(* CODESYS project Ergasia.project

Project tree, tasks and I/O mapping:
  Device : CODESYS Control Win V3, 3S - Smart Software Solutions GmbH, version 3.5.3.50
    application Application
      libraries: Standard, 3.5.2.0 (System)
      task MainTask (cyclic, interval t#20ms, priority 1) calls Main, Simulate
      task VISU_TASK (cyclic, interval 100 ms, priority 30) calls VisuElems.Visu_Prg
      program Main [SFC]: machine_check, Turn_off
      global variables GVL
      function block Flow_Control [SFC]: try_load, reset
      program Simulate [ST]
      visualisation Visualization
  text list GlobalTextList
  GlobalImagePool
*)

// Device/Application/GVL
VAR_GLOBAL
	start_switch: BOOL;
	stop_switch: BOOL;
	load_bottle: BOOL;
	water_filler: BOOL;
	water_filler_time: LREAL := 5;
	water_filler_end: BOOL;
	wf_elapsed: LREAL;
	bottle_position: LREAL;
	water_filler_lens: BOOL;
	capper_lens: BOOL;
	tagger_lens: BOOL;
	storing_bank_lens: BOOL := FALSE;
	corridor_moving: BOOL;
	capper_end: BOOL;
	tagger_time: LREAL := 3;
	tagger_end: BOOL;
	capper: BOOL;
	tagger: BOOL;
	capper_elapsed: LREAL;
	tagger_elapsed: LREAL;
	capper_time: LREAL := 2;
	stop_button: BOOL := FALSE;
	bottle_number: INT := 0;
	supplying_bank_lens: BOOL := TRUE;
	stbl_on_time: LREAL := 0;
	alarm: BOOL := FALSE;
	running: BOOL;
	full_supplying_bank: BOOL := FALSE;
	finished_bottles: INT := 0;
END_VAR

// Device/Application/Main
PROGRAM Main
VAR
	succ_check: BOOL;
END_VAR

VAR
	Flow_Control: Flow_Control;
END_VAR

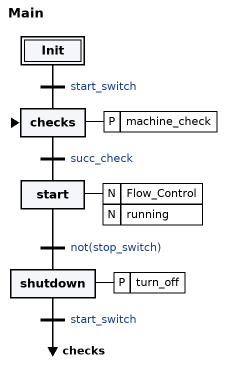
INITIAL_STEP Init:
END_STEP
TRANSITION FROM Init TO checks
    := start_switch;
END_TRANSITION
STEP checks:
    machine_check(P);
END_STEP
TRANSITION FROM checks TO start
    := succ_check;
END_TRANSITION
STEP start:
    Flow_Control(N);
    running(N);
END_STEP
TRANSITION FROM start TO shutdown
    := not(stop_switch);
END_TRANSITION
STEP shutdown:
    turn_off(P);
END_STEP
TRANSITION FROM shutdown TO checks
    := start_switch;
END_TRANSITION

ACTION machine_check:
IF (NOT(corridor_moving) AND NOT(water_filler) AND NOT(capper) AND NOT(tagger)) THEN
	succ_check := TRUE;
END_IF
END_ACTION

ACTION Turn_off:
(* calculate remaining time of operations *)
(*water_filler_time := water_filler_time - wf_elapsed;
capper_time := capper_time - capper_elapsed;
tagger_time := tagger_time - tagger_elapsed;*)
(*shut down machines *)
corridor_moving := FALSE;
water_filler := FALSE;
capper := FALSE;
tagger := FALSE;
succ_check := FALSE;
END_ACTION

END_PROGRAM

// Device/Application/Flow_Control
FUNCTION_BLOCK Flow_Control
VAR_INPUT
END_VAR
VAR_OUTPUT
END_VAR
VAR
END_VAR

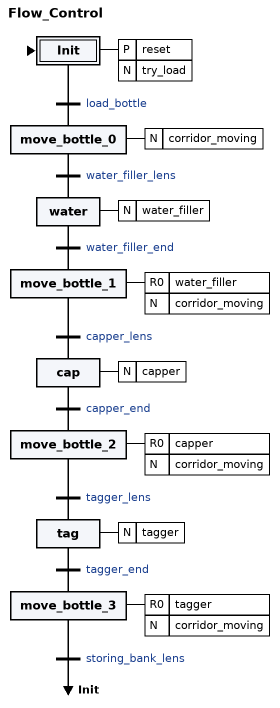
INITIAL_STEP Init:
    reset(P);
    try_load(N);
END_STEP
TRANSITION FROM Init TO move_bottle_0
    := load_bottle;
END_TRANSITION
STEP move_bottle_0:
    corridor_moving(N);
END_STEP
TRANSITION FROM move_bottle_0 TO water
    := water_filler_lens;
END_TRANSITION
STEP water:
    water_filler(N);
END_STEP
TRANSITION FROM water TO move_bottle_1
    := water_filler_end;
END_TRANSITION
STEP move_bottle_1:
    water_filler(R0);
    corridor_moving(N);
END_STEP
TRANSITION FROM move_bottle_1 TO cap
    := capper_lens;
END_TRANSITION
STEP cap:
    capper(N);
END_STEP
TRANSITION FROM cap TO move_bottle_2
    := capper_end;
END_TRANSITION
STEP move_bottle_2:
    capper(R0);
    corridor_moving(N);
END_STEP
TRANSITION FROM move_bottle_2 TO tag
    := tagger_lens;
END_TRANSITION
STEP tag:
    tagger(N);
END_STEP
TRANSITION FROM tag TO move_bottle_3
    := tagger_end;
END_TRANSITION
STEP move_bottle_3:
    tagger(R0);
    corridor_moving(N);
END_STEP
TRANSITION FROM move_bottle_3 TO Init
    := storing_bank_lens;
END_TRANSITION

ACTION try_load:
IF bottle_number > 0 AND supplying_bank_lens = TRUE THEN
	load_bottle := TRUE;
ELSE
	load_bottle := FALSE;
END_IF
END_ACTION

ACTION reset:
water_filler_end := FALSE;
capper_end := FALSE;
tagger_end := FALSE;
bottle_position := 0;
END_ACTION

END_FUNCTION_BLOCK

// Device/Application/Simulate
PROGRAM Simulate
VAR
END_VAR

(* initially closed switch simulation *)
stop_switch := NOT(stop_button);

(* completed bottle_number bottles simulation *)
IF bottle_number = 0 AND running THEN
	stop_button := TRUE;
END_IF

(* empty supplying bank simulation *)
IF supplying_bank_lens = FALSE AND bottle_position = 0 AND bottle_number > 0 THEN
	stop_button := TRUE;
	alarm := TRUE;
END_IF
IF supplying_bank_lens = TRUE AND bottle_position = 0 AND bottle_number > 0 THEN
	stop_button := FALSE;
	alarm := FALSE;
END_IF

(* full storing bank simulation *)
IF storing_bank_lens = TRUE AND full_supplying_bank THEN
	storing_bank_lens := TRUE;
ELSIF storing_bank_lens = TRUE AND NOT(full_supplying_bank) THEN
	storing_bank_lens := FALSE;
	stop_button := FALSE;
	alarm := FALSE;
	stbl_on_time := 0;
END_IF
IF storing_bank_lens = TRUE AND bottle_number > 0 THEN
	stbl_on_time := stbl_on_time + 0.02;
	IF stbl_on_time >= 2 THEN (* 2s lens on - arbitrary value *)
		stop_button := TRUE;
		alarm := TRUE;
	END_IF
END_IF

(* bottle moving in corridor simulation *)
IF (corridor_moving) THEN
	wf_elapsed := 0;
	capper_elapsed := 0;
	tagger_elapsed := 0;
	water_filler_lens := FALSE;
	capper_lens := FALSE;
	tagger_lens := FALSE;
	bottle_position := bottle_position + 0.015;
	IF bottle_position >=3 AND bottle_position <3.1 THEN
		water_filler_lens := TRUE;
		bottle_position := 3.2;
	ELSIF bottle_position >=6.1 AND bottle_position <6.2 THEN
		capper_lens := TRUE;
		bottle_position := 6.2;
	ELSIF bottle_position >=9.2 AND bottle_position <9.3 THEN
		tagger_lens := TRUE;
		bottle_position :=9.3;
	ELSIF bottle_position >=12.3 AND bottle_position <12.4 THEN
		storing_bank_lens := TRUE;
		bottle_position := 12.4;
		bottle_number := bottle_number - 1; (* bottle is finished *)
		finished_bottles := finished_bottles + 1;
	END_IF
END_IF

(* watering machine simulation *)
IF (water_filler) THEN
	water_filler_lens := TRUE;
	wf_elapsed := wf_elapsed + 0.02; (* 20ms cycle *)
	IF wf_elapsed >= water_filler_time THEN
		water_filler_end := TRUE;
	END_IF
END_IF

(* capping machine simulation *)
IF (capper) THEN
	capper_lens := TRUE;
	capper_elapsed := capper_elapsed + 0.02; (* 20ms cycle *)
	IF capper_elapsed >= capper_time THEN
		capper_end := TRUE;
	END_IF
END_IF

(* tagging machine simulation *)
IF (tagger) THEN
	tagger_lens := TRUE;
	tagger_elapsed := tagger_elapsed + 0.02; (* 20ms cycle *)
	IF tagger_elapsed >= tagger_time THEN
		tagger_end := TRUE;
	END_IF
END_IF

END_PROGRAM

// Device/Application/Visualization
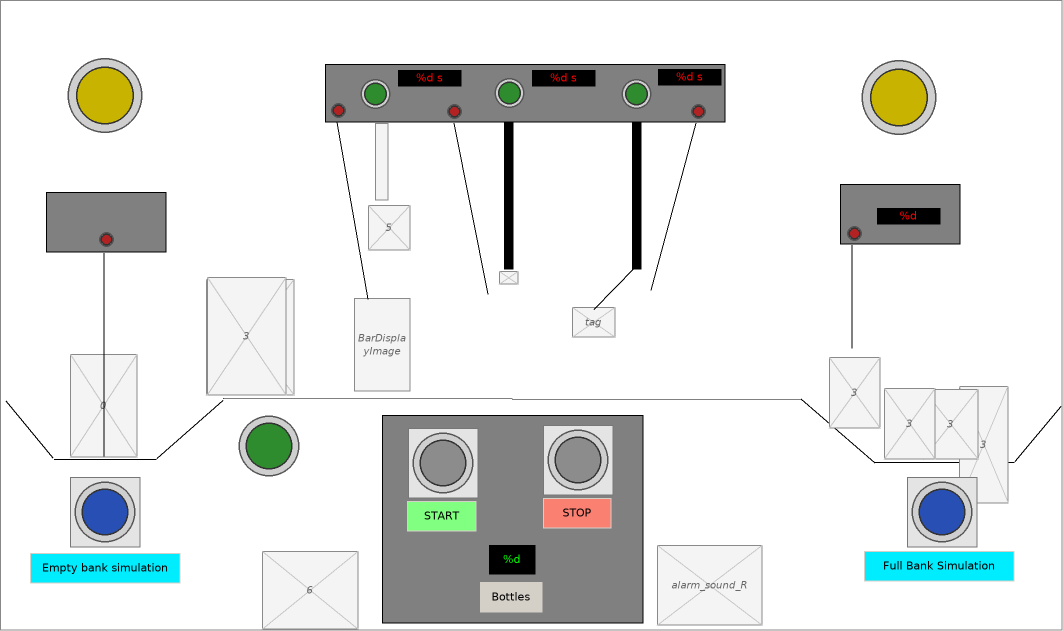
VISUALIZATION Visualization  // 1063x631
    Rectangle (382,415 261x208)
    PushSwitch (408,428 70x70), variable: start_switch, behaviour: TAP, style: Switch-PushSwitch-Gray
    PushSwitch (543,425 70x70), variable: stop_button, behaviour: TAP, style: Switch-PushSwitch-Gray
    Rectangle (489,545 46x29), "%d", text variable: bottle_number
        OnMouseDown: write the text variable via Edit, min 0, max 999
    Line (223,398) (801,399)
    Rectangle (325,64 400x58)
    BarDisplayImage (354,298 56x93), value: wf_elapsed, style: BarDisplayImage-Gray, scale format: %.1f, scale 0..5
    BarDisplayImage (375,123 13x77), value: 5-wf_elapsed, style: BarDisplayImage-Yellow, scale format: %.1f, scale 0..5
    Image (208,278 74x114), invisible if: water_filler_end, image: 0
        p3560616238: 42*bottle_position
    Image (207,283 74x111), invisible if: not(water_filler_end) or capper_end, image: 1
        p3560616238: 42*(bottle_position)
    Rectangle (504,122 9x147)
    Image (499,271 19x13), invisible if: not(capper), image: 2
    Image (206,279 88x116), invisible if: not(capper_end) or tagger_end, image: 4
        p3560616238: 42*bottle_position
    Rectangle (632,122 9x147)
    Image (572,307 43x30), invisible if: not(tagger), image: tag
    Line (594,309) (635,267), invisible if: not(tagger)
    Image (207,277 79x118), invisible if: not(tagger_end), image: 3
        p3560616238: 42*bottle_position
    Lamp1 (358,77 35x34), variable: water_filler, style: Lamp-Lamp1-Green
    Lamp1 (492,76 35x34), variable: capper, style: Lamp-Lamp1-Green
    Lamp1 (619,77 35x34), variable: tagger, style: Lamp-Lamp1-Green
    Lamp1 (328,102 21x17), variable: water_filler_lens, style: Lamp-Lamp1-Red
    Line (368,299) (337,122)
    Lamp1 (444,103 21x17), variable: capper_lens, style: Lamp-Lamp1-Red
    Lamp1 (688,103 21x17), variable: tagger_lens, style: Lamp-Lamp1-Red
    Line (488,294) (454,123)
    Line (651,290) (696,123)
    Image (368,205 42x45), invisible if: not(water_filler), image: 5
    Line (875,463) (801,399)
    Line (875,462) (1014,462)
    Line (1015,461) (1061,406)
    Line (53,458) (6,401)
    Line (54,459) (156,459)
    Line (157,458) (223,400)
    Image (959,386 49x117), invisible if: finished_bottles < 1, image: 3
    Image (923,389 55x70), invisible if: finished_bottles < 2, image: 3
    Image (884,388 51x71), invisible if: finished_bottles < 3, image: 3
    Rectangle (840,184 120x60)
    Lamp1 (844,225 21x17), variable: storing_bank_lens, style: Lamp-Lamp1-Red
    Line (852,348) (852,245)
    Rectangle (46,192 120x60)
    Lamp1 (96,231 21x17), variable: supplying_bank_lens, style: Lamp-Lamp1-Red
    Line (104,356) (104,253)
    Image (70,354 67x103), invisible if: not(supplying_bank_lens), image: 0
    PushSwitch (70,477 70x70), variable: supplying_bank_lens, behaviour: TOGGLE, style: Switch-PushSwitch-Blue
    PushSwitch (907,477 70x70), variable: full_supplying_bank, behaviour: TOGGLE, style: Switch-PushSwitch-Blue
    Textfield (30,553 150x30), "Empty bank simulation"
    Textfield (864,551 150x30), "Full Bank Simulation"
    Line (104,456) (104,353), invisible if: supplying_bank_lens
    Lamp1 (61,52 88x87), variable: alarm, style: Lamp-Lamp1-Yellow
    Lamp1 (855,54 88x87), variable: alarm, style: Lamp-Lamp1-Yellow
    Image (829,357 51x71), invisible if: stbl_on_time < 2, image: 3
    Textfield (407,501 69x30), "START"
    Textfield (543,498 68x30), "STOP"
    Textfield (480,582 62x30), "Bottles"
    Textfield (398,70 63x16), "%d s", text variable: wf_elapsed
    Textfield (532,70 63x16), "%d s", text variable: capper_elapsed
    Textfield (658,69 63x16), "%d s", text variable: tagger_elapsed
    Textfield (877,208 63x16), "%d", text variable: finished_bottles
    Image (262,551 96x78), invisible if: not(alarm), image: 6
    Image (657,545 105x80), invisible if: not(alarm), image: alarm_sound_R
    Lamp1 (234,411 70x70), variable: corridor_moving, style: Lamp-Lamp1-Green
END_VISUALIZATION
